{attribute 'GeneratedUsingTerminal: EL2521-0124-0016'}
{attribute addProperty BoxType "EL2521-0124-0016"}
{attribute addProperty Id "Sel_Ack_End_counterAT %I*BOOL1Ramp_activeAT %I*BOOL1ErrorAT %I*BOOL1Sync_ErrorAT %I*BOOL1TxPDO_ToggleAT %I*BOOL1"}
{attribute addProperty CRC "3335777329"}
{attribute addProperty Size "5"}
TYPE PTO_Status_C6D3EC31 :
STRUCT
	{attribute addProperty Name "Sel_Ack_End_counter"}
	Sel_Ack_End_counter AT %I* : BOOL;
	{attribute addProperty Name "Ramp_active"}
	Ramp_active AT %I* : BOOL;
	{attribute addProperty Name "Error"}
	Error AT %I* : BOOL;
	{attribute addProperty Name "Sync_Error"}
	Sync_Error AT %I* : BOOL;
	{attribute addProperty Name "TxPDO_Toggle"}
	TxPDO_Toggle AT %I* : BOOL;
END_STRUCT
END_TYPE

(* stored: Version 1.2.0.0, ProductVersion 3.1.4024.9
   DUT PTO_Status_C6D3EC31: Id {b4c5cb42-738e-4d13-9692-9751af96cf27} *)
